FUNCTION TryConvert_ULINT_TO_DATE : BOOL
VAR_INPUT
	in : ULINT;
	out : REFERENCE TO DATE;
END_VAR

IF in > DatatypeLimits.MAX_VALUE_OF_ULINT_WHICH_CAN_BE_HELD_IN_A_DATE THEN
	RETURN;
END_IF

out := ULINT_TO_DATE(in);
TryConvert_ULINT_TO_DATE := TRUE;

END_FUNCTION

(* stored: Version 1.1.0.1, ProductVersion 3.1.4024.12
   POU TryConvert_ULINT_TO_DATE: Id {084180e8-362f-4f2a-be9b-0c5f4b922de4}, SpecialFunc None *)
